FUNCTION_BLOCK P_Wait (* Timer event: EO after DT; RESET cancels *)
  (* Standard: 61499-2 *)
  (* Version 2.0, 2026-09-27, Project contributors, Filling cell reference model *)
  PACKAGE fillingcell;
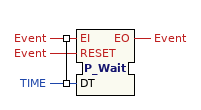
  EVENT_INPUT
    EI WITH DT;
    RESET;
  END_EVENT
  EVENT_OUTPUT
    EO;
  END_EVENT
  VAR_INPUT
    DT : TIME := T#1s;
  END_VAR
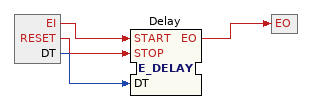
  FBS
    Delay : iec61499::events::E_DELAY;
  END_FBS
  EVENT_CONNECTIONS
    EI TO Delay.START;
    RESET TO Delay.STOP;
    Delay.EO TO EO;
  END_CONNECTIONS
  DATA_CONNECTIONS
    DT TO Delay.DT;
  END_CONNECTIONS
END_FUNCTION_BLOCK
